// SIMATIC S7-200 project (STEP 7-Micro/WIN), CPU 224 REL 02.01

SYMBOL_TABLE 用户定义1
起动               I0.0
停止               I0.1
一号呼车             I0.2
二号呼车             I0.3
三号呼车             I0.4
四号呼车             I0.5
五号呼车             I0.6
一号工位             I0.7
二号工位             I1.0
三号工位             I1.1
四号工位             I1.2
五号工位             I1.3
正转               Q0.0
反转               Q0.1
可以呼车             Q0.2
小车启停控制           M0.0
END_SYMBOL_TABLE

SYMBOL_TABLE S7-200 符号
Always_On        SM0.0    // 始终接通为 ON
Pot0_Value       SMB28    // 包含与模拟电位器 0 对应的数值
END_SYMBOL_TABLE

ORGANIZATION_BLOCK 主程序:OB1
TITLE=程序注释
BEGIN
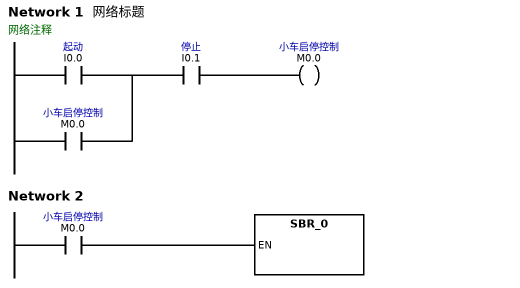
Network 1 // 网络标题
// 网络注释
LD     起动:I0.0
O      小车启停控制:M0.0
A      停止:I0.1
=      小车启停控制:M0.0
Network 2
LD     小车启停控制:M0.0
CALL   SBR_0:SBR0
END_ORGANIZATION_BLOCK

SUBROUTINE_BLOCK SBR_0:SBR0
TITLE=小车呼车控制
BEGIN
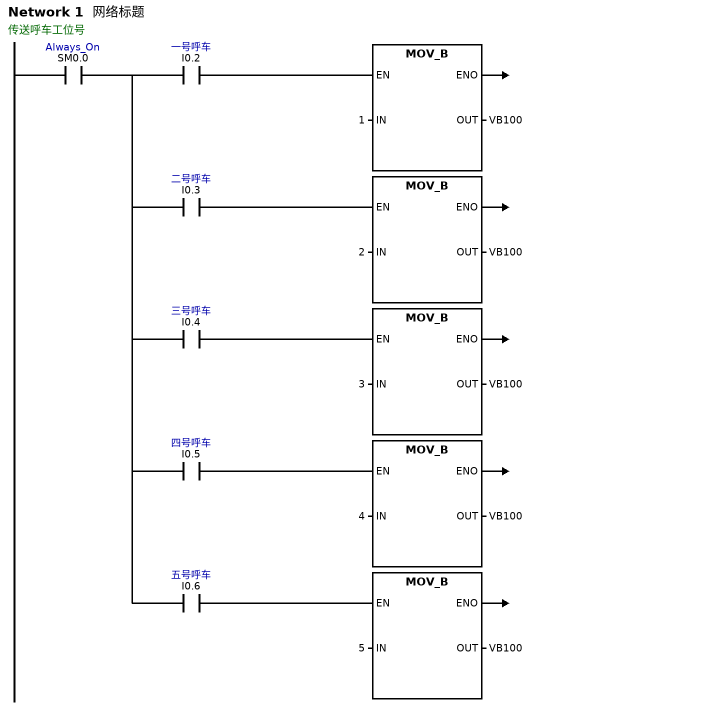
Network 1 // 网络标题
// 传送呼车工位号
LD     Always_On:SM0.0
LPS
A      一号呼车:I0.2
MOVB   1, VB100
LRD
A      二号呼车:I0.3
MOVB   2, VB100
LRD
A      三号呼车:I0.4
MOVB   3, VB100
LRD
A      四号呼车:I0.5
MOVB   4, VB100
LPP
A      五号呼车:I0.6
MOVB   5, VB100
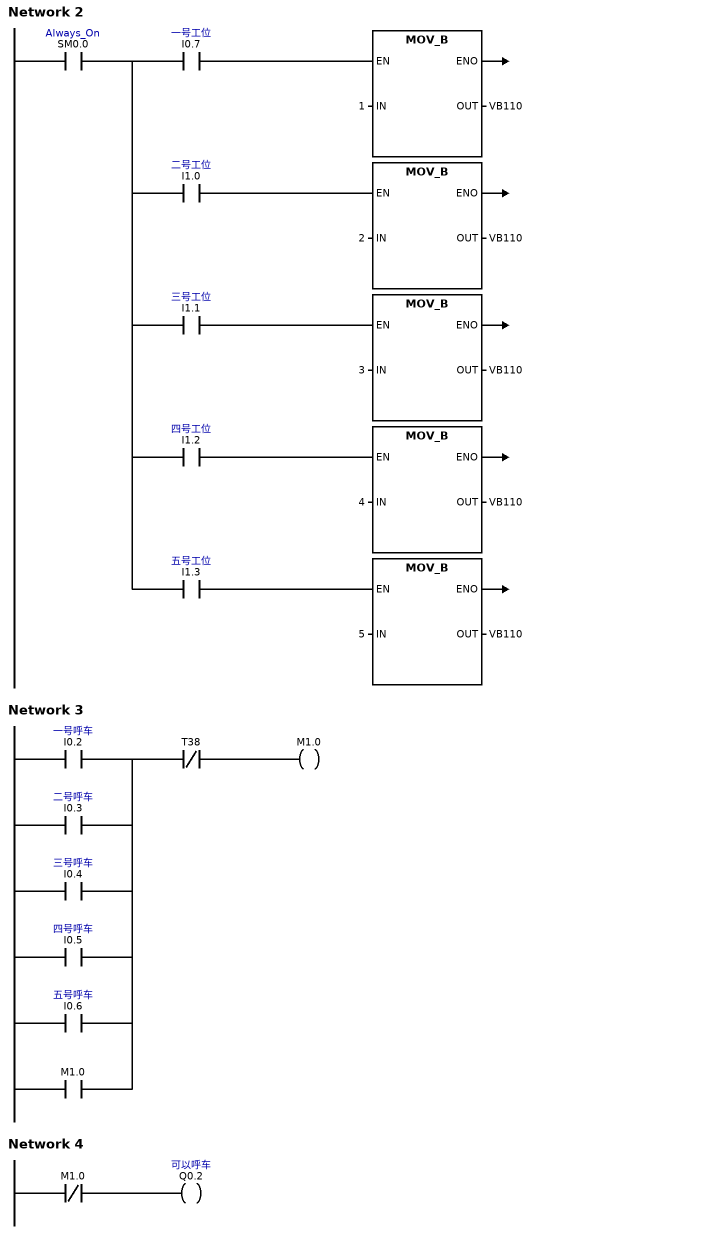
Network 2
LD     Always_On:SM0.0
LPS
A      一号工位:I0.7
MOVB   1, VB110
LRD
A      二号工位:I1.0
MOVB   2, VB110
LRD
A      三号工位:I1.1
MOVB   3, VB110
LRD
A      四号工位:I1.2
MOVB   4, VB110
LPP
A      五号工位:I1.3
MOVB   5, VB110
Network 3
LD     一号呼车:I0.2
O      二号呼车:I0.3
O      三号呼车:I0.4
O      四号呼车:I0.5
O      五号呼车:I0.6
O      M1.0
AN     T38
=      M1.0
Network 4
LDN    M1.0
=      可以呼车:Q0.2
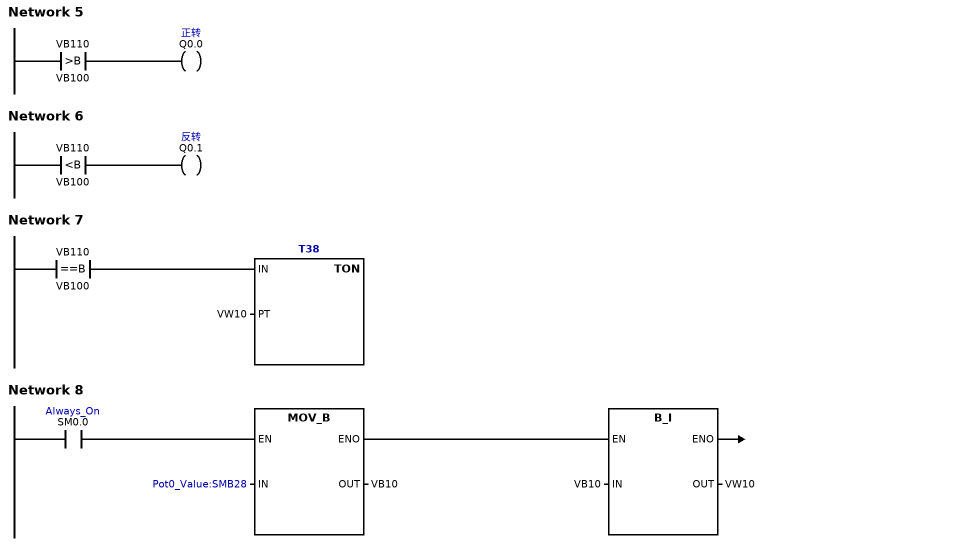
Network 5
LDB>   VB110, VB100
=      正转:Q0.0
Network 6
LDB<   VB110, VB100
=      反转:Q0.1
Network 7
LDB=   VB110, VB100
TON    T38, VW10
Network 8
LD     Always_On:SM0.0
MOVB   Pot0_Value:SMB28, VB10
AENO
BTI    VB10, VW10
END_SUBROUTINE_BLOCK
